// TIA Portal V17 export
// export: Created 2025-07-01T14:25:46.0102005Z, ExportSetting WithDefaults, DisplayName Totally Integrated Automation Portal, DisplayVersion V17 Update 8, DisplayName TIA Portal Openness, DisplayVersion V17 Update 8, DisplayName TIA Portal Version Control Interface, DisplayVersion V17, DisplayName SINAMICS Startdrive Advanced, DisplayVersion V17 SP2, DisplayName SINAMICS Startdrive G110M, G120, G120C, G120D, G120P, G115D, DisplayVersion V17 SP2, DisplayName SINAMICS Startdrive G130, G150, S120, S150, SINAMICS MV, S210, DisplayVersion V17 SP2, DisplayName STEP 7 Professional, DisplayVersion V17 Update 8, DisplayName SINUMERIK ONE STEP 7 Toolbox, DisplayVersion V17 Update 12, DisplayName SINUMERIK ONE PLC Basic Program Plus, DisplayVersion V17 Update 12, DisplayName SINUMERIK 840D sl STEP 7 Toolbox, DisplayVersion V17 Update 12, DisplayName STEP 7 Safety, DisplayVersion V17 Update 6, DisplayName WinCC Advanced, DisplayVersion V17 Update 8
FUNCTION "FC2007_INCREMENTAL_MODE" : Void   // FC2007, LAD
{ S7_Optimized_Access := 'FALSE' }
AUTHOR : ETXETAR
VERSION : 1.0
// stored: AutoNumber false, IsIECCheckEnabled false, SetENOAutomatically false, UDAEnableTagReadback false
   VAR CONSTANT
      FC_NUMBER : DInt := 2014;
   END_VAR
BEGIN

REGION Network 1: CALL FB2007 MG1
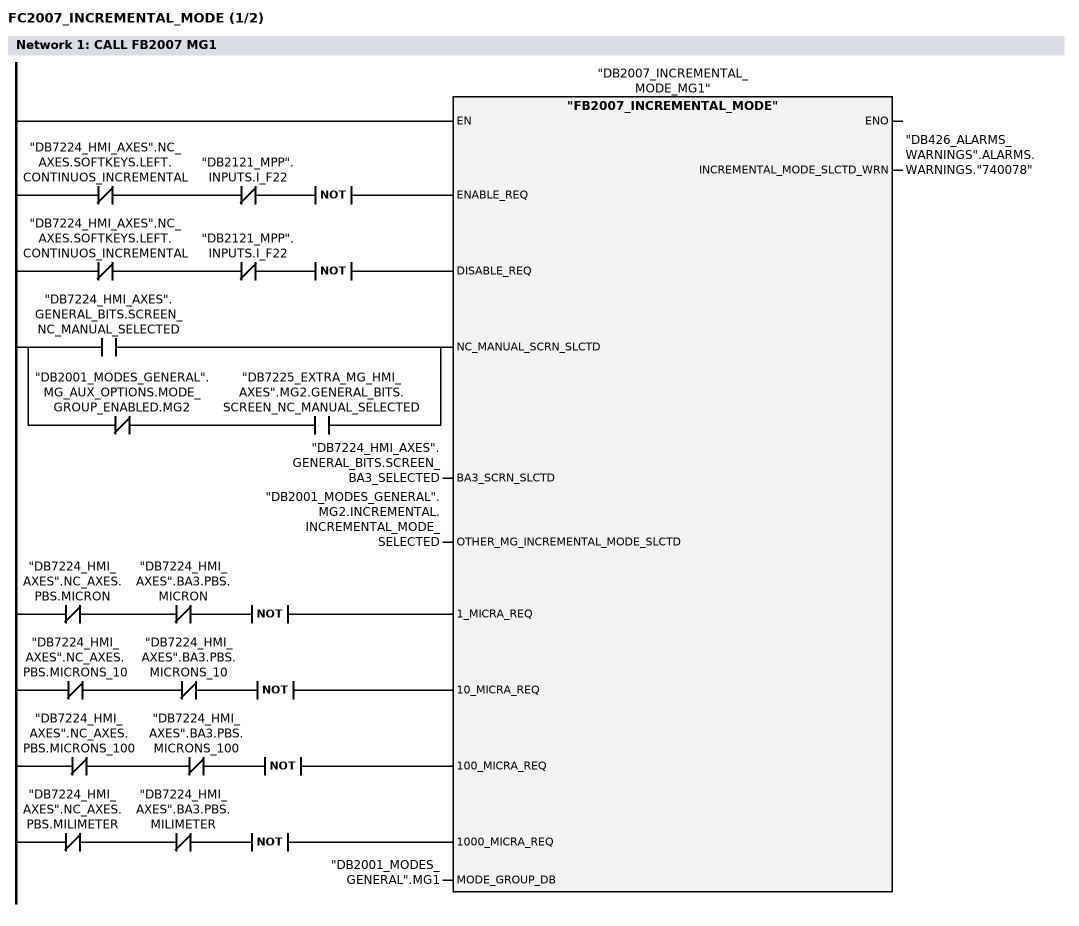
   RUNG wire#powerrail
      "DB2007_INCREMENTAL_MODE_MG1"(ENABLE_REQ := wire#w1, DISABLE_REQ := wire#w2, NC_MANUAL_SCRN_SLCTD := wire#w3, "1_MICRA_REQ" := wire#w4, "10_MICRA_REQ" := wire#w5, "100_MICRA_REQ" := wire#w6, "1000_MICRA_REQ" := wire#w7, BA3_SCRN_SLCTD := "DB7224_HMI_AXES".GENERAL_BITS.SCREEN_BA3_SELECTED, OTHER_MG_INCREMENTAL_MODE_SLCTD := "DB2001_MODES_GENERAL".MG2.INCREMENTAL.INCREMENTAL_MODE_SELECTED, MODE_GROUP_DB := "DB2001_MODES_GENERAL".MG1, INCREMENTAL_MODE_SLCTD_WRN => "DB426_ALARMS_WARNINGS".ALARMS.WARNINGS."740078")
   END_RUNG
   RUNG wire#powerrail
      I_Contact( "DB7224_HMI_AXES".NC_AXES.SOFTKEYS.LEFT.CONTINUOS_INCREMENTAL )
      I_Contact( "DB2121_MPP".INPUTS.I_F22 )
      Not()
   END_RUNG wire#w1
   RUNG wire#powerrail
      I_Contact( "DB7224_HMI_AXES".NC_AXES.SOFTKEYS.LEFT.CONTINUOS_INCREMENTAL )
      I_Contact( "DB2121_MPP".INPUTS.I_F22 )
      Not()
   END_RUNG wire#w2
   RUNG wire#powerrail
      Contact( "DB7224_HMI_AXES".GENERAL_BITS.SCREEN_NC_MANUAL_SELECTED )
   END_RUNG wire#w3
   RUNG wire#powerrail
      I_Contact( "DB2001_MODES_GENERAL".MG_AUX_OPTIONS.MODE_GROUP_ENABLED.MG2 )
      Contact( "DB7225_EXTRA_MG_HMI_AXES".MG2.GENERAL_BITS.SCREEN_NC_MANUAL_SELECTED )
   END_RUNG wire#w3
   RUNG wire#powerrail
      I_Contact( "DB7224_HMI_AXES".NC_AXES.PBS.MICRON )
      I_Contact( "DB7224_HMI_AXES".BA3.PBS.MICRON )
      Not()
   END_RUNG wire#w4
   RUNG wire#powerrail
      I_Contact( "DB7224_HMI_AXES".NC_AXES.PBS.MICRONS_10 )
      I_Contact( "DB7224_HMI_AXES".BA3.PBS.MICRONS_10 )
      Not()
   END_RUNG wire#w5
   RUNG wire#powerrail
      I_Contact( "DB7224_HMI_AXES".NC_AXES.PBS.MICRONS_100 )
      I_Contact( "DB7224_HMI_AXES".BA3.PBS.MICRONS_100 )
      Not()
   END_RUNG wire#w6
   RUNG wire#powerrail
      I_Contact( "DB7224_HMI_AXES".NC_AXES.PBS.MILIMETER )
      I_Contact( "DB7224_HMI_AXES".BA3.PBS.MILIMETER )
      Not()
   END_RUNG wire#w7
   // the same network as SCL:
   "DB2007_INCREMENTAL_MODE_MG1"(ENABLE_REQ := NOT (NOT "DB7224_HMI_AXES".NC_AXES.SOFTKEYS.LEFT.CONTINUOS_INCREMENTAL AND NOT "DB2121_MPP".INPUTS.I_F22),   // "FB2007_INCREMENTAL_MODE"
                           DISABLE_REQ := NOT (NOT "DB7224_HMI_AXES".NC_AXES.SOFTKEYS.LEFT.CONTINUOS_INCREMENTAL AND NOT "DB2121_MPP".INPUTS.I_F22),
                           NC_MANUAL_SCRN_SLCTD := "DB7224_HMI_AXES".GENERAL_BITS.SCREEN_NC_MANUAL_SELECTED OR (NOT "DB2001_MODES_GENERAL".MG_AUX_OPTIONS.MODE_GROUP_ENABLED.MG2 AND "DB7225_EXTRA_MG_HMI_AXES".MG2.GENERAL_BITS.SCREEN_NC_MANUAL_SELECTED),
                           BA3_SCRN_SLCTD := "DB7224_HMI_AXES".GENERAL_BITS.SCREEN_BA3_SELECTED,
                           OTHER_MG_INCREMENTAL_MODE_SLCTD := "DB2001_MODES_GENERAL".MG2.INCREMENTAL.INCREMENTAL_MODE_SELECTED,
                           "1_MICRA_REQ" := NOT (NOT "DB7224_HMI_AXES".NC_AXES.PBS.MICRON AND NOT "DB7224_HMI_AXES".BA3.PBS.MICRON),
                           "10_MICRA_REQ" := NOT (NOT "DB7224_HMI_AXES".NC_AXES.PBS.MICRONS_10 AND NOT "DB7224_HMI_AXES".BA3.PBS.MICRONS_10),
                           "100_MICRA_REQ" := NOT (NOT "DB7224_HMI_AXES".NC_AXES.PBS.MICRONS_100 AND NOT "DB7224_HMI_AXES".BA3.PBS.MICRONS_100),
                           "1000_MICRA_REQ" := NOT (NOT "DB7224_HMI_AXES".NC_AXES.PBS.MILIMETER AND NOT "DB7224_HMI_AXES".BA3.PBS.MILIMETER),
                           MODE_GROUP_DB := "DB2001_MODES_GENERAL".MG1,
                           INCREMENTAL_MODE_SLCTD_WRN => "DB426_ALARMS_WARNINGS".ALARMS.WARNINGS."740078");
END_REGION

REGION Network 2: CALL FB2007 MG2
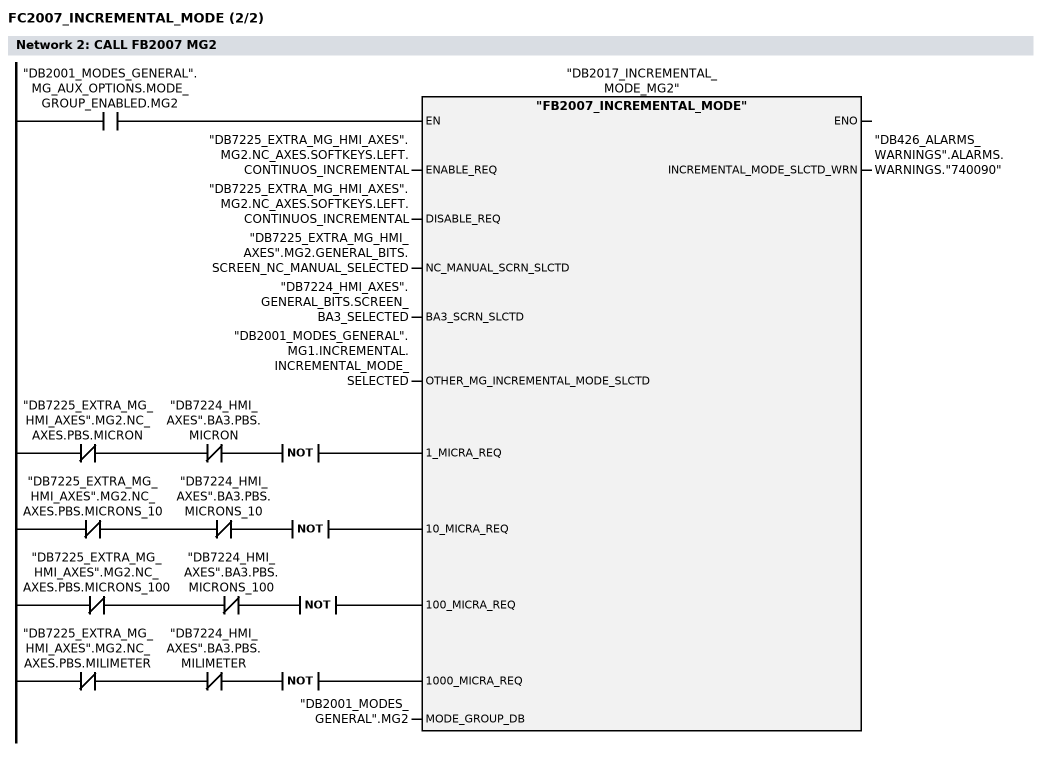
   RUNG wire#powerrail
      Contact( "DB2001_MODES_GENERAL".MG_AUX_OPTIONS.MODE_GROUP_ENABLED.MG2 )
      "DB2017_INCREMENTAL_MODE_MG2"("1_MICRA_REQ" := wire#w1, "10_MICRA_REQ" := wire#w2, "100_MICRA_REQ" := wire#w3, "1000_MICRA_REQ" := wire#w4, ENABLE_REQ := "DB7225_EXTRA_MG_HMI_AXES".MG2.NC_AXES.SOFTKEYS.LEFT.CONTINUOS_INCREMENTAL, DISABLE_REQ := "DB7225_EXTRA_MG_HMI_AXES".MG2.NC_AXES.SOFTKEYS.LEFT.CONTINUOS_INCREMENTAL, NC_MANUAL_SCRN_SLCTD := "DB7225_EXTRA_MG_HMI_AXES".MG2.GENERAL_BITS.SCREEN_NC_MANUAL_SELECTED, BA3_SCRN_SLCTD := "DB7224_HMI_AXES".GENERAL_BITS.SCREEN_BA3_SELECTED, OTHER_MG_INCREMENTAL_MODE_SLCTD := "DB2001_MODES_GENERAL".MG1.INCREMENTAL.INCREMENTAL_MODE_SELECTED, MODE_GROUP_DB := "DB2001_MODES_GENERAL".MG2, INCREMENTAL_MODE_SLCTD_WRN => "DB426_ALARMS_WARNINGS".ALARMS.WARNINGS."740090")
   END_RUNG
   RUNG wire#powerrail
      I_Contact( "DB7225_EXTRA_MG_HMI_AXES".MG2.NC_AXES.PBS.MICRON )
      I_Contact( "DB7224_HMI_AXES".BA3.PBS.MICRON )
      Not()
   END_RUNG wire#w1
   RUNG wire#powerrail
      I_Contact( "DB7225_EXTRA_MG_HMI_AXES".MG2.NC_AXES.PBS.MICRONS_10 )
      I_Contact( "DB7224_HMI_AXES".BA3.PBS.MICRONS_10 )
      Not()
   END_RUNG wire#w2
   RUNG wire#powerrail
      I_Contact( "DB7225_EXTRA_MG_HMI_AXES".MG2.NC_AXES.PBS.MICRONS_100 )
      I_Contact( "DB7224_HMI_AXES".BA3.PBS.MICRONS_100 )
      Not()
   END_RUNG wire#w3
   RUNG wire#powerrail
      I_Contact( "DB7225_EXTRA_MG_HMI_AXES".MG2.NC_AXES.PBS.MILIMETER )
      I_Contact( "DB7224_HMI_AXES".BA3.PBS.MILIMETER )
      Not()
   END_RUNG wire#w4
   // the same network as SCL:
   IF "DB2001_MODES_GENERAL".MG_AUX_OPTIONS.MODE_GROUP_ENABLED.MG2 THEN
       "DB2017_INCREMENTAL_MODE_MG2"(ENABLE_REQ := "DB7225_EXTRA_MG_HMI_AXES".MG2.NC_AXES.SOFTKEYS.LEFT.CONTINUOS_INCREMENTAL,   // "FB2007_INCREMENTAL_MODE"
                               DISABLE_REQ := "DB7225_EXTRA_MG_HMI_AXES".MG2.NC_AXES.SOFTKEYS.LEFT.CONTINUOS_INCREMENTAL,
                               NC_MANUAL_SCRN_SLCTD := "DB7225_EXTRA_MG_HMI_AXES".MG2.GENERAL_BITS.SCREEN_NC_MANUAL_SELECTED,
                               BA3_SCRN_SLCTD := "DB7224_HMI_AXES".GENERAL_BITS.SCREEN_BA3_SELECTED,
                               OTHER_MG_INCREMENTAL_MODE_SLCTD := "DB2001_MODES_GENERAL".MG1.INCREMENTAL.INCREMENTAL_MODE_SELECTED,
                               "1_MICRA_REQ" := NOT (NOT "DB7225_EXTRA_MG_HMI_AXES".MG2.NC_AXES.PBS.MICRON AND NOT "DB7224_HMI_AXES".BA3.PBS.MICRON),
                               "10_MICRA_REQ" := NOT (NOT "DB7225_EXTRA_MG_HMI_AXES".MG2.NC_AXES.PBS.MICRONS_10 AND NOT "DB7224_HMI_AXES".BA3.PBS.MICRONS_10),
                               "100_MICRA_REQ" := NOT (NOT "DB7225_EXTRA_MG_HMI_AXES".MG2.NC_AXES.PBS.MICRONS_100 AND NOT "DB7224_HMI_AXES".BA3.PBS.MICRONS_100),
                               "1000_MICRA_REQ" := NOT (NOT "DB7225_EXTRA_MG_HMI_AXES".MG2.NC_AXES.PBS.MILIMETER AND NOT "DB7224_HMI_AXES".BA3.PBS.MILIMETER),
                               MODE_GROUP_DB := "DB2001_MODES_GENERAL".MG2,
                               INCREMENTAL_MODE_SLCTD_WRN => "DB426_ALARMS_WARNINGS".ALARMS.WARNINGS."740090");
   END_IF;
END_REGION
END_FUNCTION
